// Core §3.10.2 — one configuration value served through the request mailbox
// instead of the cyclic OPC UA tree. Scope selects the owner ('' = the root
// Unit itself, a qualified dotted module identity for a child, '#Fieldbus' for
// the bus topology). Item is the value's browse fragment in the server's array
// naming (e.g. 'Catalog/Catalog[2]/Label') so a generic HMI can rebuild the
// exact published path it would otherwise have read.
TYPE ST_ConfigEntry :
STRUCT
    Scope     : STRING(255);
    Item      : STRING(255);
    ValueText : STRING(255);   // typed by the HMI from the Item vocabulary
END_STRUCT
END_TYPE

(* stored: Version 1.1.0.1, ProductVersion 3.1.4024.12
   DUT ST_ConfigEntry: Id {8f3d92a1-6c47-4b0e-9d15-2a7e84c1f603} *)
